FUNCTION_BLOCK FB_PIDControl (* Basic Function Block Type *)
  (* Standard: 61499-2 *)
  (* Version 0.0, 2014-5-4, wildai, nxtControl GmbH, Template *)
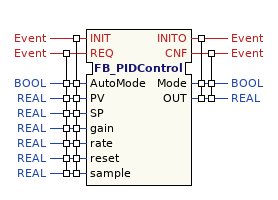
  EVENT_INPUT
    INIT WITH AutoMode, PV, SP, gain, rate, reset, sample; (* Initialization Request *)
    REQ WITH AutoMode, PV, SP, gain, rate, reset, sample; (* Normal Execution Request *)
  END_EVENT
  EVENT_OUTPUT
    INITO WITH Mode, OUT; (* Initialization Confirm *)
    CNF WITH Mode, OUT; (* Execution Confirmation *)
  END_EVENT
  VAR_INPUT
    AutoMode : BOOL;
    PV : REAL;
    SP : REAL;
    gain : REAL;
    rate : REAL;
    reset : REAL;
    sample : REAL;
  END_VAR
  VAR_OUTPUT
    Mode : BOOL;
    OUT : REAL;
  END_VAR
  VAR
    SPin : REAL;
    PVscl : REAL;
    SPscl : REAL;
    OUTscl : REAL;
    error : REAL;
    bias : REAL;
    PVold : REAL;
    I_Coeff : REAL;
    D_Coeff : REAL;
    curMode : BOOL;
    firstCycle : BOOL;
    Mp : REAL;
    Mi : REAL;
    Md : REAL;
    Ma : REAL;
  END_VAR
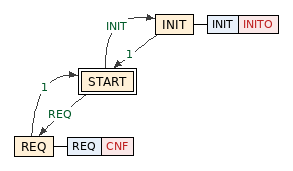
  EC_STATES
    START; (* Initial State *)
    INIT : INIT -> INITO; (* Initialization *)
    REQ : REQ -> CNF; (* Normal execution *)
  END_STATES
  EC_TRANSITIONS
    START TO INIT := INIT;
    INIT TO START := 1;
    START TO REQ := REQ;
    REQ TO START := 1;
  END_TRANSITIONS
  ALGORITHM INIT IN ST: (* Initialization algorithm *)
;

Mode := FALSE;
OUT := 0.0;
  END_ALGORITHM
  ALGORITHM REQ IN ST: (* Normally executed algorithm *)
;

/* Precalculate PID cofeeicients */
I_Coeff := 0.0;
SPin := SP;
IF reset <> 0 THEN
	I_Coeff := sample / reset;
END_IF;
D_Coeff := rate / sample;

/* Multiply I, D cofficeints by gain if gain is used */
IF gain <> 0 THEN
	I_Coeff := I_Coeff * gain;
	D_Coeff := D_Coeff * gain;
END_IF;

/* Auto -> Manual Transition */
IF ((NOT AutoMode) AND curMode) THEN
	firstCycle := TRUE;
	curMode := FALSE;
	Mode := FALSE;
/* Manual -> Auto Transition */
ELSIF (AutoMode AND (NOT curMode)) THEN
	bias := OUT / 27648;
	SPin := PV;
	firstCycle := TRUE;
	curMode := TRUE;
	Mode := TRUE;
END_IF;

IF curMode THEN
	/*Scale PV if > 100% then clamp at 100%, if PV < 0% then clamp to 0% */
	IF PV <= 0 THEN
		PVscl := 0.0;
	ELSIF PV > 27648 THEN
		PVscl := 1.0;
	ELSE
		PVscl := PV / 27648;
	END_IF;

	/* Scale Setpoint if SP > 100% then clamp to 100%, if SP < 0% then clamp to 0% */
	IF SPin < 0 THEN
		SPscl := 0.0;
	ELSIF SPin >= 27648 THEN
		SPscl := 1.0;
	ELSE
		SPscl := SPin / 27648;
	END_IF;

	/* Calculate Error */
	error := SPin - PV;
	/* Calculate PID terms */
	Mp := gain * error;
	Mi := bias + (I_Coeff * error);
	Md := 0.0;

	/* If derivative used then calculate Md */
	IF ((rate <> 0) AND (NOT firstCycle)) THEN
		Md := D_Coeff * (PVold - PV);
	END_IF;

	/* Calcuulate provisional output (before bias clamping) */
	PVold := PVscl;
	Ma := Mp + Md;
	OUT := Ma + Mi;

	/* Bias Clamping: if Output > 100%, clamp and backcalculate bias */
	IF OUT > 1 THEN
		OUTscl := 1.0;
		Mi := 1.0 - Ma;
	ELSIF OUT < 0 THEN
		OUTscl := 0.0;
		Mi := 0.0 - Ma;
	END_IF;

	/* Clamp bias to 0 to 1 range */
	IF I_Coeff <> 0.0 THEN
		IF Mi > 1.0 THEN
			Mi := 1.0;
		ELSIF Mi < 0.0 THEN
			Mi := 0.0;
		ELSE
			bias := Mi;
		END_IF;
	END_IF;

	/* Reset first cycle flag and unscale output */
	firstCycle := FALSE;
	OUT := OUTscl * 27648;
END_IF;
  END_ALGORITHM
END_FUNCTION_BLOCK
